(* IEC 61131-3 sources: tutorials/projects/ch07-2/PROGRAM, 1 file *)

(* ---- main_prog.st ---- *)
PROGRAM PLC_PRG
    VAR
        // INPUTS [0..2]对应modbus寄存器12,13,14读入数值
        // OUTPUTS[0..2]对应要写入modbus寄存器12,13,14的数值
        // OUTPUTS AT %QB12 : ARRAY[0..2] OF BYTE;
        // INPUTS AT %IB12 : ARRAY[0..2] OF BYTE;

        // INPUT10_0 AT %IX10.0: BOOL;
        // INPUT10_1 AT %IX10.1: BOOL;

        // ERR_CNT: 对应modbus寄存器20, 用来输出错误计数
        // ERR_CNT AT %QW20 : INT := 1;

        i : INT := 0;
        cur : INT := -1;
    END_VAR

    // x0, x1, x2：在IO表中配置的输入全局变量，对应modbus寄存器1, 2, 4
    // t0, t1, t2：在IO表中配置的输出全局变量，对应modbus寄存器100, 101, 103
    // 在IO表中以上变量的IO内存位置设置为“自动”，由IDE自动分配

    // 测试python会写入modbus寄存器1, 2, 4，然后读取modbus寄存器100, 101, 103
    // 使用读取的数值对比写入的数值来验证ST在工作正常

    // 设置t0为x0+1
    t0 := x0 + 1;

    // 设置t1为x1-1
    t1 := x1 - 1;

    // 设置t2等于x2
    t2 := x2;

    //WARNING('cur: %d, INPUT10.1:%d, INPUT10.1: %d', cur, TO_INT(INPUT10_1), TO_INT(INPUT10_1));

    // 忽略第一个周期
    IF cur = -1 THEN
        cur := 0;
    ELSE
        // 验证在modbus寄存器12..14本周期读出来的值等于上周期写入的值
        FOR i:= 0 TO 2 DO
            IF INPUTS[i] <> OUTPUTS[i] THEN
                ERR_CNT := ERR_CNT + 1;
                WA_LOG('Mismatch - %d', i);
            END_IF
        END_FOR;
    END_IF;

    WARNING('#%d, INPUTS:[%d,%d,%d]', cur, INPUTS[0], INPUTS[1],INPUTS[2]);

    // 对于modbus寄存器12..14进行跑马灯写值
   FOR i:= 0 TO 2 DO
       OUTPUTS[i]:= INPUTS[i];
   END_FOR;
   INPUTS[cur] := 1;

   cur := cur + 1;
    IF cur = 3 THEN
        cur := 0;
    END_IF;

   WARNING('#%d, OUTPUTS:[%d,%d,%d]', cur, OUTPUTS[0], OUTPUTS[1],OUTPUTS[2]);

END_PROGRAM
